(* Logix 5000 project; controller Ex_2_18 Emulate 5570 rev 33.11; software revision 33.00 *)
// Conveyor for pallet pickup (Man/Auto)

TASK MainTask (continuous, watchdog 500 ms) : MainProgram

MODULES
   Local : Emulate 5570 (ICP 4, rev 33.11)
END_MODULES

VAR_GLOBAL   (* controller tags *)
   B1 : BOOL;   // Sensor B1
   Conveyor_Operation : BOOL;
   M1 : BOOL;   // Conveyor_Running
   P1 : BOOL;   // Lamp P1
   P2 : BOOL;   // Lamp P2
   S1 : BOOL;   // Switch S1
   S2_Auto_Mode : BOOL;
   S3 : BOOL;   // S3_Man_PB
   S3_Man_Mode : BOOL;
END_VAR

PROGRAM MainProgram   (* main routine MainRoutine *)

ROUTINE MainRoutine   (* ladder *)
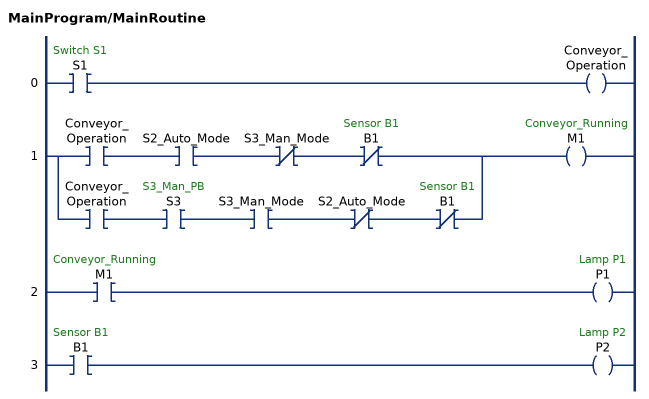
   0: XIC(S1)OTE(Conveyor_Operation);
   1: [XIC(Conveyor_Operation) XIC(S2_Auto_Mode) XIO(S3_Man_Mode) XIO(B1) ,XIC(Conveyor_Operation) XIC(S3) XIC(S3_Man_Mode) XIO(S2_Auto_Mode) XIO(B1) ]OTE(M1);
   2: XIC(M1)OTE(P1);
   3: XIC(B1)OTE(P2);
END_ROUTINE
END_PROGRAM
